FUNCTION_BLOCK PUBLIC PAEEmergencySwitch EXTENDS PAESensorDigital
VAR_INPUT
END_VAR
VAR_OUTPUT
END_VAR
VAR
END_VAR

END_FUNCTION_BLOCK

(* stored: Version 1.1.0.1, ProductVersion 3.1.4020.6
   POU PAEEmergencySwitch: Id {f4a2c1fb-11f8-445b-945f-9b171d7646a5}, SpecialFunc None *)
